PROGRAM MAIN
VAR
END_VAR

DoorControlLogic();

END_PROGRAM

(* stored: Version 1.1.0.1, ProductVersion 3.1.4022.18
   POU MAIN: Id {30828e1c-e934-40bb-9799-4da1a38f5c46}, SpecialFunc None *)
